ABB RobotStudio station: 2. undervisning_20200306-062353.rsstn

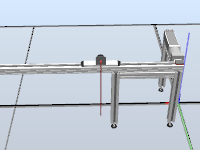
Station 2. undervisning (saved by RobotStudio 7.0.8728.594)
Layout (positions relative to the parent item):
  - base_2 [part] at (0, 0, -80) mm, rotated rx 90 ry 0 rz 0 deg
  - cart_2 [part] at (83.94, -25, 445) mm, rotated rx 90 ry 0 rz 0 deg
  - Part_3 [part]
  - pendul [part] at (483.94, 239.5, 480) mm, rotated rx 90 ry 0 rz 0 deg
  - Part_8 [part]
  - Part_9 [part]
